FUNCTION_BLOCK InfluentFeed (* CAT Function Block Type *)
  (* Standard: 61499-2 *)
  (* Version 0.0, 13/09/2026, template *)
  PACKAGE Hidryco.HidrycoLib;
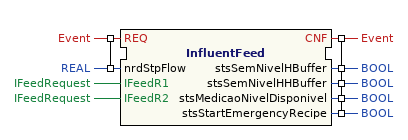
  EVENT_INPUT
    REQ WITH nrdStpFlow;
  END_EVENT
  EVENT_OUTPUT
    CNF WITH stsSemNivelHBuffer, stsSemNivelHHBuffer, stsMedicaoNivelDisponivel, stsStartEmergencyRecipe;
  END_EVENT
  VAR_INPUT
    nrdStpFlow : REAL;
  END_VAR
  VAR_OUTPUT
    stsSemNivelHBuffer : BOOL;
    stsSemNivelHHBuffer : BOOL;
    stsMedicaoNivelDisponivel : BOOL;
    stsStartEmergencyRecipe : BOOL;
  END_VAR
  SOCKETS
    IFeedR1 : IFeedRequest;
    IFeedR2 : IFeedRequest;
  END_SOCKETS
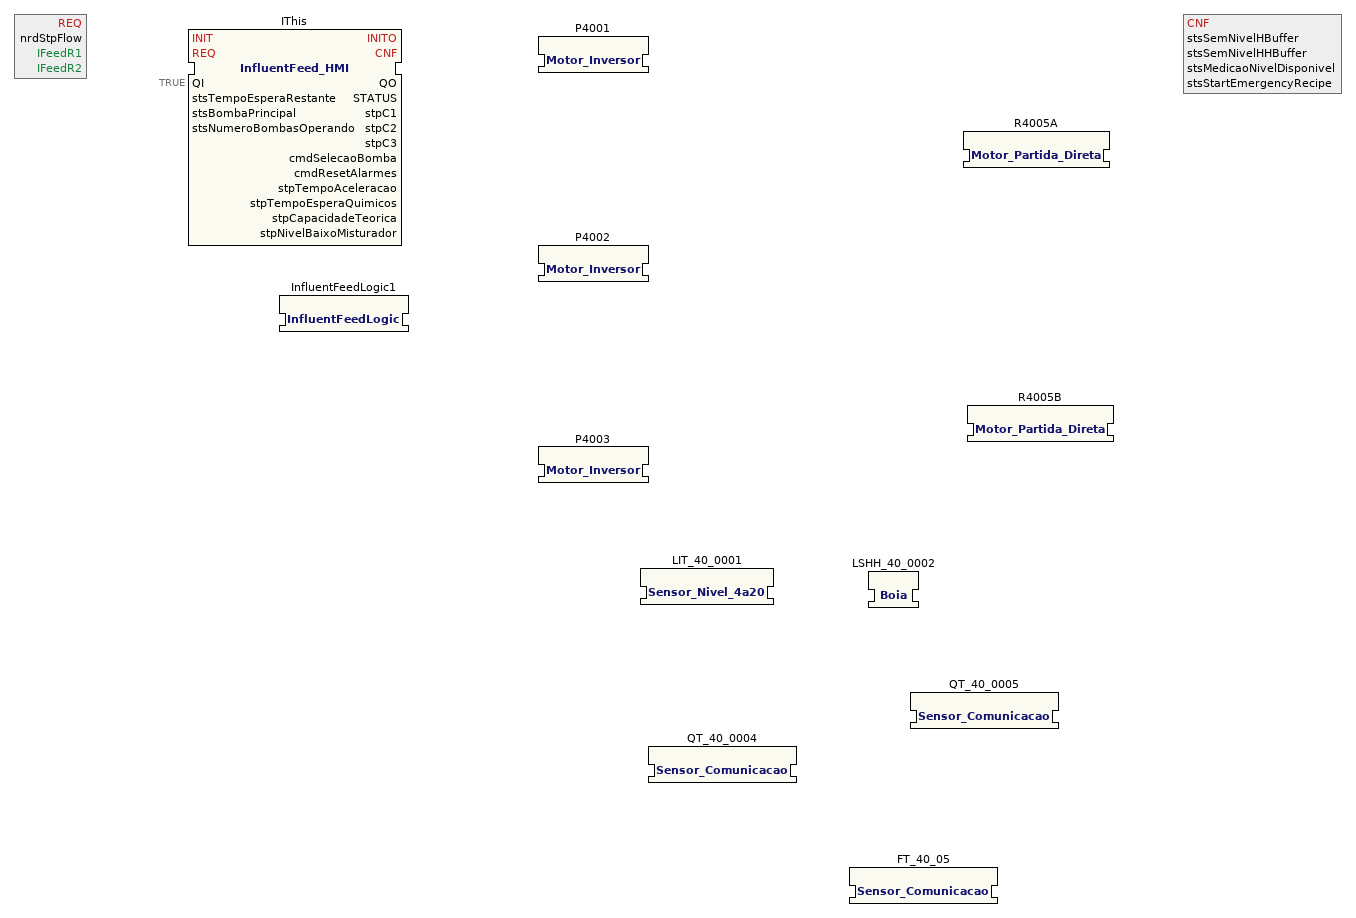
  (* Atudores *)
  (* Sensores *)
  FBS
    IThis : InfluentFeed_HMI(QI := TRUE);
    P4001 : Motor_Inversor;
    P4002 : Motor_Inversor;
    P4003 : Motor_Inversor;
    R4005A : Motor_Partida_Direta;
    R4005B : Motor_Partida_Direta;
    LIT_40_0001 : Sensor_Nivel_4a20;
    LSHH_40_0002 : Boia;
    QT_40_0004 : Sensor_Comunicacao;
    QT_40_0005 : Sensor_Comunicacao;
    FT_40_05 : Sensor_Comunicacao;
    InfluentFeedLogic1 : InfluentFeedLogic;
  END_FBS
END_FUNCTION_BLOCK
